{attribute 'qualified_only'}
{attribute 'strict'}
TYPE DUT_ENUM :
(
	enum_member := 0,
	OFF,
	ON
);
END_TYPE

(* stored: Version 1.1.0.1, ProductVersion 3.1.4024.4
   DUT DUT_ENUM: Id {b79a7a58-b3e4-490e-8ea2-636b29c84889} *)
